Staubli VAL3: Move.pgx

program Move()
begin
  resetMotion()
  while !bExit
    nWorkingMode=workingMode(nStatus)
    if nWorkingMode==1 and nStatus==0
      movel(pFrameRefPt[nSelectedPt],tTool,mNomSpeed)
      waitEndMove()
    else
      resetMotion()
    endIf
    delay(0)
  endWhile
  resetMotion()
end
